FUNCTION IntegerBitAccess : BOOL
VAR_INPUT
	num : ULINT;
	n : ULINT;
END_VAR

IntegerBitAccess := (SHR(num, n) AND 1) > 0;

END_FUNCTION

(* stored: Version 1.1.0.1, ProductVersion 3.1.4024.11
   POU IntegerBitAccess: Id {b06922ad-687f-4f20-8c5d-74dac39fd7e3}, SpecialFunc None *)
